(* IEC 61131-3 sources: Lasal/CPU_5344_V01/Class/ScreenCtrl, 1 file *)

(* ---- ScreenCtrl.st ---- *)
(*!
<Class
	Name               = "ScreenCtrl"
	Revision           = "0.0"
	RealtimeTask       = "false"
	CyclicTask         = "false"
	BackgroundTask     = "true"
	DefBackground      = "1000 ms"
	Sigmatek           = "false"
	OSInterface        = "false"
	HighPriority       = "false"
	Automatic          = "false"
	UpdateMode         = "Prescan"
	SharedCommandTable = "true"
	Objectsize         = "(450,360)">
	<Channels>
		<Server Name="ActScreen" Visualized="true" Initialize="false" WriteProtected="false" Retentive="false"/>
		<Server Name="ActWindow" Visualized="true" Initialize="false" WriteProtected="false" Retentive="false"/>
		<Server Name="ClassSvr" Visualized="false" Initialize="false" WriteProtected="true" Retentive="false"/>
		<Server Name="CloseWindow" Visualized="true" Initialize="false" WriteProtected="false" Retentive="false"/>
		<Server Name="dateValue" Visualized="true" Initialize="false" WriteProtected="false" Retentive="false"/>
		<Server Name="NrAlarms" Visualized="true" Initialize="false" WriteProtected="false" Retentive="false"/>
		<Server Name="ProgChangeAllowed" Visualized="true" Initialize="false" WriteProtected="false" Retentive="false"/>
		<Server Name="ReqScreen" Visualized="true" Initialize="false" WriteProtected="false" Retentive="false"/>
		<Server Name="ReqWindow" Visualized="true" Initialize="false" WriteProtected="false" Retentive="false"/>
		<Server Name="syncTime" Visualized="false" Initialize="true" DefValue="1" WriteProtected="false" Retentive="false"/>
		<Server Name="timeValue" Visualized="true" Initialize="false" WriteProtected="false" Retentive="false"/>
		<Server Name="UserLevel" Visualized="true" Initialize="false" WriteProtected="false" Retentive="false"/>
		<Client Name="ctrlDateTime" Required="true" Internal="false"/>
		<Client Name="updateDate" Required="true" Internal="false"/>
		<Client Name="updateTime" Required="true" Internal="false"/>
	</Channels>
</Class>
*)
ScreenCtrl : CLASS
  //Servers:
	ClassSvr 	: SvrChCmd_DINT;
	ActScreen 	: SvrCh_DINT;
	ActWindow 	: SvrCh_DINT;
	ReqScreen 	: SvrCh_DINT;
	ReqWindow 	: SvrCh_DINT;
	CloseWindow 	: SvrCh_DINT;
	NrAlarms 	: SvrCh_DINT;
	UserLevel 	: SvrCh_DINT;
	ProgChangeAllowed 	: SvrCh_DINT;
	timeValue 	: SvrCh_HDINT;
	dateValue 	: SvrCh_HDINT;
	syncTime 	: SvrCh_DINT;
  //Clients:
	ctrlDateTime 	: CltChCmd__SysDateTime2;
	updateTime 	: CltCh_HDINT;
	updateDate 	: CltCh_HDINT;
  //Variables:
		oldTimeValue 	: HDINT;
		oldDateValue 	: HDINT;
  //Functions:

	FUNCTION VIRTUAL GLOBAL Init;

	FUNCTION VIRTUAL GLOBAL Background
		VAR_INPUT
			EAX 	: UDINT;
		END_VAR
		VAR_OUTPUT
			state (EAX) 	: UDINT := READY;
		END_VAR;
  //Tables:
	FUNCTION @STD
		VAR_OUTPUT
			ret_code	: CONFSTATES;
		END_VAR;
	FUNCTION GLOBAL TAB @CT_;
END_CLASS;

#pragma usingLtd _SysDateTime2

// JdK 27-11-2019: ScreenCtrl class to copy values from kernel project to cpu project and other way around
// added function to sync time with time of screen project

FUNCTION VIRTUAL GLOBAL ScreenCtrl::Init

  ReqScreen := ReqWindow :=UserLevel := -1;
  timeValue:= 0;
  dateValue:= 0;

END_FUNCTION

FUNCTION VIRTUAL GLOBAL ScreenCtrl::Background
	VAR_INPUT
		EAX 	: UDINT;
	END_VAR
	VAR_OUTPUT
		state (EAX) 	: UDINT;(* := READY *)
	END_VAR

  //sync date and time with visualisation
  IF syncTime THEN
    IF dateValue<> 0 & timeValue <> 0 & (oldTimeValue<> timeValue | oldDateValue<> dateValue) THEN //time and date value are written from kernel project
      IF timeValue <> ctrlDateTime.SysTime THEN //only write update if they are not the same
        updateTime.Write(input:=timeValue);
      END_IF;
      IF dateValue <> ctrlDateTime.SysDate THEN
        updateDate.Write(input:=dateValue);
      END_IF;
      oldTimeValue:= timeValue;
      oldDateValue:= dateValue;
    END_IF;
  END_IF;

END_FUNCTION
